ABB RobotStudio station: Exam.rsstn

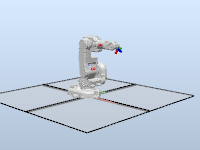
Station Exam (saved by RobotStudio 20.4.9280.0)
Layout (positions relative to the parent item):
  - IRB140_6_81_C_03 [mechanism, from Robots\IRB140_6_81_C_G_03.rslib] at (0, 0, 0) mm; joint values [0, 0, 0, 0, 0.5236, 0] (rad or m)
